// Internal class that manages the ITcIecApplicationInfo TcCOM Interface used by Fs_Standard.
{attribute 'no_assign'}
{attribute 'no_explicit_call' := 'direct call for this function block is not allowed'} 
FUNCTION_BLOCK INTERNAL FINAL FsFB_TcComIecApplicationInfo IMPLEMENTS FsI_UnKnown
VAR
	_ipIecApplicationInformation : ITcIecApplicationInfo;
	_hIecApplicationInformation : HRESULT := Tc3_Module.GVL.E_FAIL;
END_VAR

{attribute 'hide'}
METHOD FB_exit : BOOL
VAR_INPUT
	bInCopyCode : BOOL; // if TRUE, the exit method is called for exiting an instance that is copied afterwards (online change).
END_VAR
// no online change
IF NOT bInCopyCode THEN
	// Safe release of ITcIecApplicationInfo.
    Tc3_Module.FW_SafeRelease(ADR(THIS^._ipIecApplicationInformation));
	THIS^._hIecApplicationInformation := Tc3_Module.GVL.E_FAIL;
	END_IF
END_METHOD

{attribute 'hide'}
{attribute 'no_explicit_call' := 'direct call for this method is not allowed'}
METHOD FB_init : BOOL
VAR_INPUT
	bInitRetains : BOOL; // if TRUE, the retain variables are initialized (warm start / cold start)
	bInCopyCode : BOOL;  // if TRUE, the instance afterwards gets moved into the copy code (online change)
END_VAR
// No online change.
IF NOT bInCopyCode THEN
	// Get instance of ITcIecApplicationInfo.
	THIS^._hIecApplicationInformation := Tc3_Module.FW_ObjMgr_GetObjectInstance(
		TwinCAT_SystemInfoVarList._AppInfo.ObjId, 
		TC_GLOBAL_IID_LIST.IID_ITcIecApplicationInfo, 
		ADR(THIS^._ipIecApplicationInformation)
	);
	END_IF
END_METHOD

METHOD GetInterface : ITcIecApplicationInfo
VAR_OUTPUT
	bSuccess : BOOL;
END_VAR
// If instance of ITcIecApplicationInfo failed to be obtained on 
// FB_init or FB_exit was explicitly called try to get it gain.
IF Tc3_Module.FAILED(THIS^._hIecApplicationInformation) THEN
	THIS^._hIecApplicationInformation := Tc3_Module.FW_ObjMgr_GetObjectInstance(
		TwinCAT_SystemInfoVarList._AppInfo.ObjId, 
		TC_GLOBAL_IID_LIST.IID_ITcIecApplicationInfo, 
		ADR(THIS^._ipIecApplicationInformation)
	);
	END_IF
	
bSuccess := Tc3_Module.SUCCEEDED(THIS^._hIecApplicationInformation);
GetInterface := THIS^._ipIecApplicationInformation;
END_METHOD

END_FUNCTION_BLOCK

(* stored: Version 1.1.0.1, ProductVersion 3.1.4024.4
   POU FsFB_TcComIecApplicationInfo: Id {e24bb523-913f-47be-9600-9bea0f20d987}, SpecialFunc None
   Method FB_exit: Id {728bc26f-a680-4b9c-8d35-54eab5f678cc}
   Method FB_init: Id {e674354e-d58d-4f55-b560-731ed7e0aaef}
   Method GetInterface: Id {33334846-ac24-44bc-aff0-c44abfe0ffa1} *)
